PROGRAM PRG_ROOTS
VAR
END_VAR

(*Roots Pump Chamber 1*)
(*gauges*)
GPI_261(PG=>);
GPI_262(PG=>);
GPI_263(PG=>);

(*Isolation Valve*)
VRC_261(Pump:=PFM_261.q_stPump,Gauge:=GPI_261.PG,i_xExtILK_OK:=TRUE);
VRC_262(Pump:=PFM_262.q_stPump,Gauge:=GPI_261.PG,i_xExtILK_OK:=TRUE);		


(* dry pump*)
PFM_261();
PFM_262();





(*Roots Pump Chamber 1*)
(*gauges*)
GPI_341(PG=>);
GPI_342(PG=>);
GPI_343(PG=>);

(*Isolation Valve*)
VRC_341(Pump:=PFM_341.q_stPump,Gauge:=GPI_341.PG,i_xExtILK_OK:=TRUE);
VRC_342(Pump:=PFM_342.q_stPump,Gauge:=GPI_341.PG,i_xExtILK_OK:=TRUE);

(* dry pump*)
PFM_341();
PFM_342();

END_PROGRAM

(* stored: Version 1.1.0.1, ProductVersion 3.1.4022.16
   POU PRG_ROOTS: Id {573f7847-bda8-45d7-9541-d46f5c27ae92}, SpecialFunc None *)
